ABB RobotStudio station: IRB1600_20220624-113841.rsstn

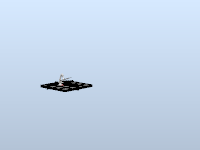
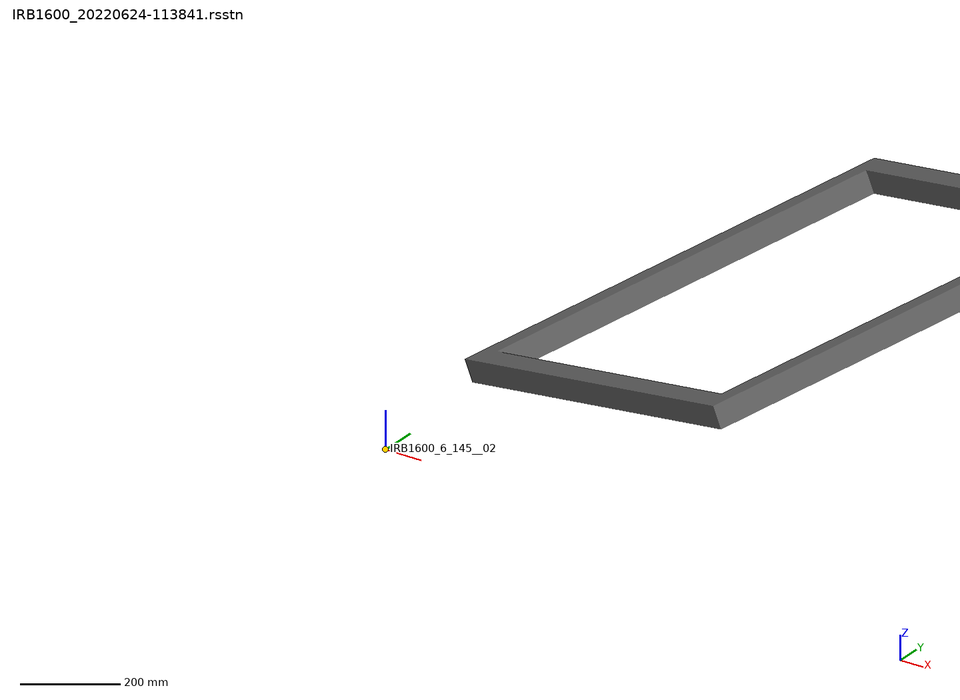
[picture v1: parts stored in the station drawn from their meshes, with robot base, taught points and paths (robot models come from the ABB library and are not in the file)]
Station Solution1 (saved by RobotStudio 22.1.9826.0)
Controller IRB1600_6_145
  mechanical unit ROB_1: IRB1600_6_145__02, 6 joints, base frame (0, 0, 0) mm
Layout (positions relative to the parent item):
  - IRB1600_6_145__02 [mechanism, from Robots\IRB1600_6_145_G_02.rslib] at (0, 0, 0) mm; joint values [-0.1388, 0.3614, 0.6216, 0.2752, -1.3034, 0.025] (rad or m)
  - flange_connector [part, from Tools\IsoPlate_small_Binzel.rslib] at (779.98, -126.13, 661.16) mm, rotated rx 30.59 ry 69.97 rz 8.3 deg
  - plane [part] at (1224.33, -321.02, 816.12) mm, rotated rx 169.49 ry 17.15 rz 156.13 deg, size 1000 x 1000 x 50 mm
  - Frame_1 [frame]
  - Frame_2 [frame] at (-23.65, -1.83, 250.36) mm
Attachment: flange_connector is attached to IRB1600_6_145__02 / Link6
Attachment: plane is attached to flange_connector
Attachment: Workobject_2 is attached to IRB1600_6_145__02 / Link1
Targets, tools, work objects and paths stored in the station, written as RAPID:
! task T_ROB1
MODULE Module1
  LOCAL PERS wobjdata egm_wobj:=[FALSE,TRUE,"",[[0,0,0],[1,0,0,0]],[[0,0,0],[1,0,0,0]]];
  TASK PERS wobjdata wobj:=[FALSE,FALSE,"ROB_1",[[639.116,-22.796,-980.437],[1,0,0,0]],[[0,0,0],[1,0,0,0]]];
  PROC main()
    ConfJ \On;
  ENDPROC
  PROC EGM_CARTESIAN_MOVE()
    WaitTime 2;
  ENDPROC
  PROC RAPID_MOVE()
  ENDPROC
ENDMODULE

! task T_ROB1
MODULE CalibData
  TASK PERS tooldata Tooldata_4:=[TRUE,[[0,0,0],[1,0,0,0]],[1,[0,0,1],[1,0,0,0],0,0,0]];
  TASK PERS tooldata Tooldata_5:=[TRUE,[[0,0,0],[1,0,0,0]],[1,[0,0,1],[1,0,0,0],0,0,0]];
  TASK PERS tooldata Tooldata_6:=[TRUE,[[0,0,0],[1,0,0,0]],[1,[0,0,1],[1,0,0,0],0,0,0]];
  TASK PERS tooldata Tooldata_7:=[TRUE,[[-23.772999698,2.161000196,740.120999999],[0.707106781,0,-0.707106781,0]],[1,[0,0,1],[1,0,0,0],0,0,0]];
  TASK PERS wobjdata Workobject_2:=[FALSE,TRUE,"",[[0,0,0],[0.997594392,0,0,-0.069321201]],[[0,0,0],[1,0,0,0]]];
  TASK PERS tooldata Tooldata_9:=[TRUE,[[20.616002648,0.899999913,497.265999882],[0.707106781,-0.000000002,-0.707106781,0]],[1,[0,0,1],[1,0,0,0],0,0,0]];
  TASK PERS wobjdata Wobj_joint1:=[TRUE,FALSE,"ROB_1",[[639.116,-613.962,-938.233],[1,0,0,0]],[[0,0,0],[1,0,0,0]]];
ENDMODULE

